Fanuc KAREL source: kt00913.KL

-- PROVISIONAL review KL for V770-1; original PC SHA256 1d0da74137e7437fe8b7c342d7d9d2eb089035a34be6a80aa71a4093871b0071
-- Incomplete behavior may be omitted. Consult companion uncertainty JSON. Do not deploy.
PROGRAM KT00913
%NOLOCKGROUP
VAR
  S1 : STRING[80]
  S2 : STRING[80]
  OUT : INTEGER
BEGIN
  -- UNRESOLVED_PC offsets 5-14; opcodes 3F,75
  -- UNRESOLVED_PC offsets 19-28; opcodes 3F,75
  -- UNRESOLVED_PC offsets 33-42; opcodes 3F,75
  -- UNRESOLVED_PC offsets 47-56; opcodes 3F,75
  -- UNRESOLVED_PC offsets 61-78; opcodes 27,22,2A,76,23
  -- UNRESOLVED_PC offsets 83-87; opcodes 7F
END KT00913
